INTERFACE I_DeserializerGarbageCollector EXTENDS __SYSTEM.IQueryInterface

METHOD PUBLIC Deregister
VAR_INPUT
	Deserializer : I_Deserializer;
END_VAR
END_METHOD

METHOD PUBLIC Register
VAR_INPUT
	Deserializer : I_Deserializer;
END_VAR
END_METHOD

END_INTERFACE

(* stored: Version 1.1.0.1, ProductVersion 3.1.4024.12
   Itf I_DeserializerGarbageCollector: Id {4a5b59bf-e662-04d9-0c1b-cefcca6186c0}
   Method Deregister: Id {ce0d799f-bb09-06e9-3df1-155e77e64d25}
   Method Register: Id {7ba8358c-e031-073e-23da-658753abf808} *)
